(* CODESYS project Trabalho_final_v2.project

Project tree, tasks and I/O mapping:
  Device : CODESYS Control Win V3, 3S - Smart Software Solutions GmbH, order no. 305021, version 3.5.11.40
    application Application
      libraries: Standard, * (System)
      task MainTask (cyclic, interval t#20ms, priority 1) calls mode_selector, flow_controller, Automatic_Tank_Controller, CoolantLevelController, flow_controller, GinFlowController, RefrigeranteFlowController, TankLevelController_T1, TankLevelController_T2, TemperatureController, VermouthFlowController, SendProductController, ConveyorControl, TonelCounter, ProductInletControl, ProductSendControl, TonelLevelControl, MixerRotationControl
      global variables GVL
      program mode_selector [LD]
      program flow_controller [SFC]: MANUAL_active, AUTOMATICO_active
      program Automatic_Tank_Controller [SFC]: Colocar_gin_active, Colocar_verm_active, Ligar_motor_active, Resfriar_active, Tirar_refrige_active, Envio_T2_active, DESATIVAR_active, REINICIAR_T1_active, Limpar_T1_active
      program TankLevelController_T1 [ST]
      program TankLevelController_T2 [ST]
      program GinFlowController [ST]
      program VermouthFlowController [ST]
      program RefrigeranteFlowController [ST]
      program TemperatureController [ST]
      program CoolantLevelController [ST]
      program SendProductController [ST]
      program ConveyorControl [SFC]: Limpa_esteira_active, Liga_esteira_active, IN_PRODU_active, Inicio_active
      program TonelCounter [ST]
      program ProductInletControl [SFC]: RETIRA_ESTEIRA_active, ABRI_TORNE_active
      program ProductSendControl [ST]
      program TonelLevelControl [ST]
      program MixerRotationControl [ST]
*)

// Device/Application/GVL
{attribute 'qualified_only'}
VAR_GLOBAL
	

	// Ativação do sistema e escolha do modo
	Ligar : BOOL := FALSE;
	EMG : BOOL := FALSE;
	Sistema_ativo: BOOL;
	Seletor: BOOL;
	Selecionado: BOOL;
	Modo_manual: BOOL;
	Modo_automatico: BOOL;
	
	
	// Ativadores de modos
	Ativador_manual: BOOL := FALSE;
	Ativador_automatico: BOOL := FALSE;
	
	// Quantidades T1
	Quantidade_total_t1 : REAL := 0;
	
	// Indicadores T1
	Tanque01_vazio : BOOL;
	Tanque01_30L : BOOL;
	Tanque01_45L : BOOL;
	Tanque01_50L : BOOL;
	
	// Quantidades de bebida
	Quantidade_total_gin : REAL := 0;
	Quantidade_total_vermouth : REAL := 0;
	Quantidade_total_refrigerante : REAL := 0;
	
	// Temporizadores bebidas
	Temporizador_entrada_gin : TON;
	Temporizador_entrada_vermouth : TON;
	Temporizador_entrada_refrigerante : TON;
	Temporizador_saida_refrigerante : TON;
	Temporizador_resfriamento : TON;
	
	// Indicadores refrigerante
	Auto_nivel_refrigerante : BOOL := FALSE;
	Baixo_nivel_refrigerante : BOOL := TRUE;
	
	// Ativador temperatura
	Ativador_temperatura : BOOL := FALSE;
	
	// Indicadores de temperatura
	Temperatura_0c : BOOL := FALSE;
	Temperatura : REAL := 27;
	
	// Quantidade t2
	Quantidade_total_t2 : REAL := 0;
	
	// Indicadores T2
	Tanque02_vazio : BOOL;
	Tanque02_10p : BOOL;
	Tanque02_50p : BOOL;
	Tanque02_85p : BOOL;
	Tanque02_95p : BOOL;
	
	//valvulas T1
	Valvula_gin : BOOL := FALSE;
	Valvula_vermouth : BOOL := FALSE;
	Valvula_refrigerante : BOOL := FALSE;
	Valvula_descarte_refrigerante : BOOL := FALSE;
	
	//Temporizadores T1
	Temporizador_descarte_produto : TON;
	Temporizador_envio_produto : TON;
	
	// Instrumentos t1
	Motor_t1 : BOOL := FALSE;
	
	// Instrumentos entre t1 e t2
	Bomba : BOOL := FALSE;
	
	// valvulas entre tanques
	Valvula_entre_tanques : BOOL := FALSE;
	Valvula_descarte : BOOL := FALSE;
	Valvula_entrada_t2 : BOOL := FALSE;
	
	//Instrumentos t2
	Esteira : BOOL;
	Termino_envio: BOOL;
	
	
	// Contadores Toneis
	Numero_toneis_liberados : REAL;
	Numero_toneis_prduzidos : REAL;
	Numero_toneis_total : REAL;
	Tonel_produzido : BOOL;
	Total_tonel_menor4: BOOL;
	Total_tonel_4: BOOL;
	
	// Temporizador produção esteira
	Temporizador_producao_esteira : TON;
	
	// Controle para o envio de produto para os toneis
	Tonel_preparado : BOOL := FALSE;
	Tonel_cheio : BOOL;
	
	// VALVULAS T2 TONEL
	Valvula_t2_tonel : BOOL := FALSE;
	Temporizador_t2_tonel : TON;
	
	//Quantidade tonel
	Quantidade_tonel : REAL;
	
	Termino_tonel : BOOL;
	Sem_produto : BOOL;
	
	// Controladores do misturador
	TON_Partida : TON;
    TON_Parada : TON;
    M101_Partida_Em_Andamento : BOOL := FALSE;
    M101_Parada_Em_Andamento : BOOL := FALSE;
	DutyCycle_OUT : REAL := 0;
END_VAR

// Device/Application/mode_selector
PROGRAM mode_selector
VAR
END_VAR

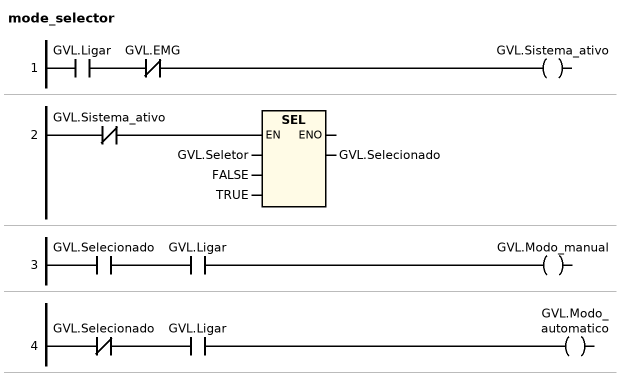
// NETWORK 1
GVL.Sistema_ativo := GVL.Ligar AND NOT GVL.EMG;

// NETWORK 2
IF NOT GVL.Sistema_ativo THEN GVL.Selecionado := SEL(GVL.Seletor, FALSE, TRUE); END_IF

// NETWORK 3
GVL.Modo_manual := GVL.Selecionado AND GVL.Ligar;

// NETWORK 4
GVL.Modo_automatico := NOT GVL.Selecionado AND GVL.Ligar;

END_PROGRAM

// Device/Application/flow_controller
PROGRAM flow_controller
VAR
END_VAR

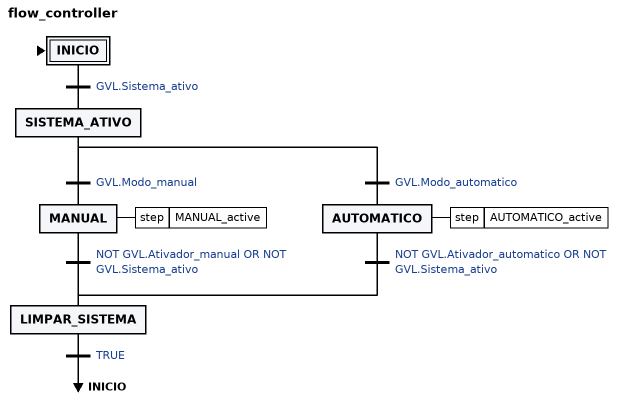
INITIAL_STEP INICIO:
END_STEP
TRANSITION FROM INICIO TO SISTEMA_ATIVO
    := GVL.Sistema_ativo;
END_TRANSITION
STEP SISTEMA_ATIVO:
END_STEP
TRANSITION FROM SISTEMA_ATIVO TO MANUAL
    := GVL.Modo_manual;
END_TRANSITION
STEP MANUAL:
    MANUAL_active(N);  // step action
END_STEP
TRANSITION FROM MANUAL TO LIMPAR_SISTEMA
    := NOT GVL.Ativador_manual OR NOT GVL.Sistema_ativo;
END_TRANSITION
TRANSITION FROM SISTEMA_ATIVO TO AUTOMATICO
    := GVL.Modo_automatico;
END_TRANSITION
STEP AUTOMATICO:
    AUTOMATICO_active(N);  // step action
END_STEP
TRANSITION FROM AUTOMATICO TO LIMPAR_SISTEMA
    := NOT GVL.Ativador_automatico OR NOT GVL.Sistema_ativo;
END_TRANSITION
STEP LIMPAR_SISTEMA:
END_STEP
TRANSITION FROM LIMPAR_SISTEMA TO INICIO
    := TRUE;
END_TRANSITION

ACTION MANUAL_active:
GVL.Ativador_manual := TRUE;
END_ACTION

ACTION AUTOMATICO_active:
GVL.Ativador_automatico := TRUE;
END_ACTION

END_PROGRAM

// Device/Application/Automatic_Tank_Controller
PROGRAM Automatic_Tank_Controller
VAR
END_VAR

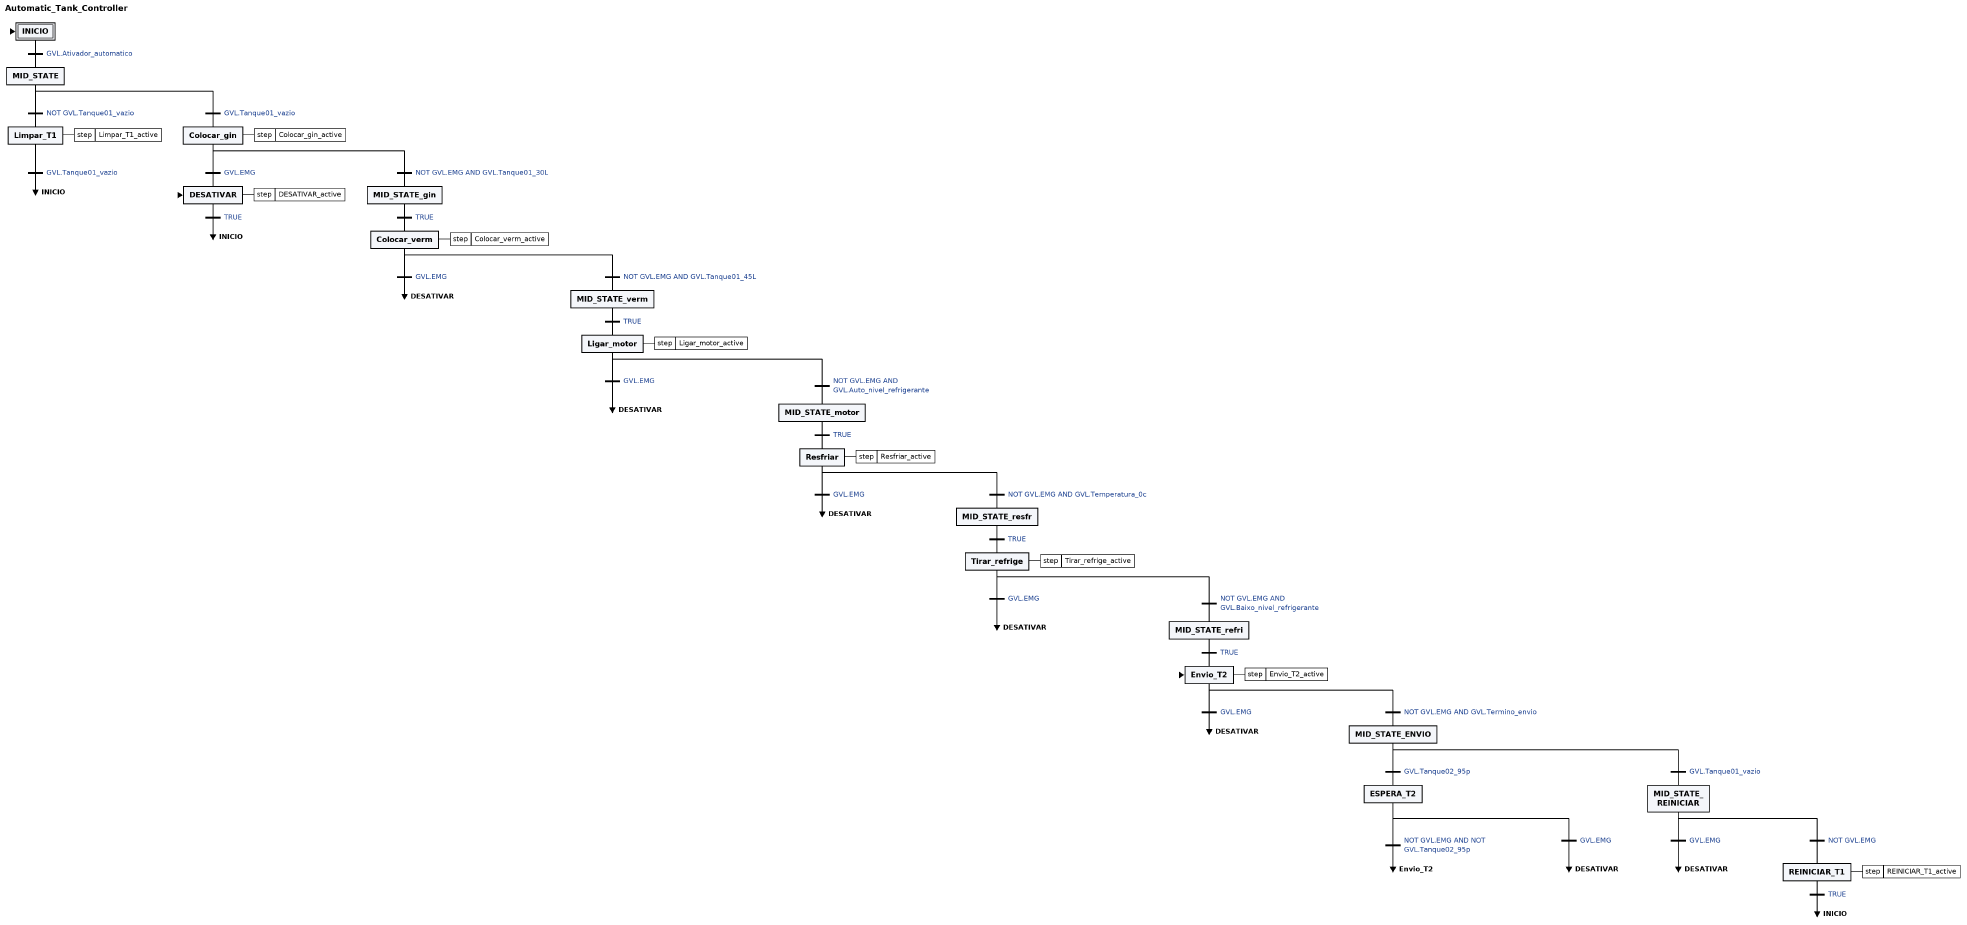
INITIAL_STEP INICIO:
END_STEP
TRANSITION FROM INICIO TO MID_STATE
    := GVL.Ativador_automatico;
END_TRANSITION
STEP MID_STATE:
END_STEP
TRANSITION FROM MID_STATE TO Limpar_T1
    := NOT GVL.Tanque01_vazio;
END_TRANSITION
STEP Limpar_T1:
    Limpar_T1_active(N);  // step action
END_STEP
TRANSITION FROM Limpar_T1 TO INICIO
    := GVL.Tanque01_vazio;
END_TRANSITION
TRANSITION FROM MID_STATE TO Colocar_gin
    := GVL.Tanque01_vazio;
END_TRANSITION
STEP Colocar_gin:
    Colocar_gin_active(N);  // step action
END_STEP
TRANSITION FROM Colocar_gin TO DESATIVAR
    := GVL.EMG;
END_TRANSITION
STEP DESATIVAR:
    DESATIVAR_active(N);  // step action
END_STEP
TRANSITION FROM DESATIVAR TO INICIO
    := TRUE;
END_TRANSITION
TRANSITION FROM Colocar_gin TO MID_STATE_gin
    := NOT GVL.EMG AND GVL.Tanque01_30L;
END_TRANSITION
STEP MID_STATE_gin:
END_STEP
TRANSITION FROM MID_STATE_gin TO Colocar_verm
    := TRUE;
END_TRANSITION
STEP Colocar_verm:
    Colocar_verm_active(N);  // step action
END_STEP
TRANSITION FROM Colocar_verm TO DESATIVAR
    := GVL.EMG;
END_TRANSITION
TRANSITION FROM Colocar_verm TO MID_STATE_verm
    := NOT GVL.EMG AND GVL.Tanque01_45L;
END_TRANSITION
STEP MID_STATE_verm:
END_STEP
TRANSITION FROM MID_STATE_verm TO Ligar_motor
    := TRUE;
END_TRANSITION
STEP Ligar_motor:
    Ligar_motor_active(N);  // step action
END_STEP
TRANSITION FROM Ligar_motor TO DESATIVAR
    := GVL.EMG;
END_TRANSITION
TRANSITION FROM Ligar_motor TO MID_STATE_motor
    := NOT GVL.EMG AND GVL.Auto_nivel_refrigerante;
END_TRANSITION
STEP MID_STATE_motor:
END_STEP
TRANSITION FROM MID_STATE_motor TO Resfriar
    := TRUE;
END_TRANSITION
STEP Resfriar:
    Resfriar_active(N);  // step action
END_STEP
TRANSITION FROM Resfriar TO DESATIVAR
    := GVL.EMG;
END_TRANSITION
TRANSITION FROM Resfriar TO MID_STATE_resfr
    := NOT GVL.EMG AND GVL.Temperatura_0c;
END_TRANSITION
STEP MID_STATE_resfr:
END_STEP
TRANSITION FROM MID_STATE_resfr TO Tirar_refrige
    := TRUE;
END_TRANSITION
STEP Tirar_refrige:
    Tirar_refrige_active(N);  // step action
END_STEP
TRANSITION FROM Tirar_refrige TO DESATIVAR
    := GVL.EMG;
END_TRANSITION
TRANSITION FROM Tirar_refrige TO MID_STATE_refri
    := NOT GVL.EMG AND GVL.Baixo_nivel_refrigerante;
END_TRANSITION
STEP MID_STATE_refri:
END_STEP
TRANSITION FROM MID_STATE_refri TO Envio_T2
    := TRUE;
END_TRANSITION
STEP Envio_T2:
    Envio_T2_active(N);  // step action
END_STEP
TRANSITION FROM Envio_T2 TO DESATIVAR
    := GVL.EMG;
END_TRANSITION
TRANSITION FROM Envio_T2 TO MID_STATE_ENVIO
    := NOT GVL.EMG AND GVL.Termino_envio;
END_TRANSITION
STEP MID_STATE_ENVIO:
END_STEP
TRANSITION FROM MID_STATE_ENVIO TO ESPERA_T2
    := GVL.Tanque02_95p;
END_TRANSITION
STEP ESPERA_T2:
END_STEP
TRANSITION FROM ESPERA_T2 TO Envio_T2
    := NOT GVL.EMG AND NOT GVL.Tanque02_95p;
END_TRANSITION
TRANSITION FROM ESPERA_T2 TO DESATIVAR
    := GVL.EMG;
END_TRANSITION
TRANSITION FROM MID_STATE_ENVIO TO MID_STATE_REINICIAR
    := GVL.Tanque01_vazio;
END_TRANSITION
STEP MID_STATE_REINICIAR:
END_STEP
TRANSITION FROM MID_STATE_REINICIAR TO DESATIVAR
    := GVL.EMG;
END_TRANSITION
TRANSITION FROM MID_STATE_REINICIAR TO REINICIAR_T1
    := NOT GVL.EMG;
END_TRANSITION
STEP REINICIAR_T1:
    REINICIAR_T1_active(N);  // step action
END_STEP
TRANSITION FROM REINICIAR_T1 TO INICIO
    := TRUE;
END_TRANSITION

ACTION Colocar_gin_active:
GVL.Valvula_gin := TRUE;
END_ACTION

ACTION Colocar_verm_active:
GVL.Valvula_vermouth := TRUE;
END_ACTION

ACTION Ligar_motor_active:
GVL.Motor_t1 := TRUE;
GVL.Valvula_refrigerante := TRUE;
END_ACTION

ACTION Resfriar_active:
GVL.Ativador_temperatura := TRUE;
END_ACTION

ACTION Tirar_refrige_active:
GVL.Motor_t1 := FALSE;
GVL.Valvula_descarte_refrigerante := TRUE;
END_ACTION

ACTION Envio_T2_active:
GVL.Valvula_entre_tanques := TRUE;
GVL.Bomba := TRUE;
GVL.Valvula_entrada_t2 := TRUE;
END_ACTION

ACTION DESATIVAR_active:
GVL.Ativador_automatico := FALSE;
END_ACTION

ACTION REINICIAR_T1_active:
GVL.Valvula_gin := FALSE;
GVL.Valvula_vermouth := FALSE;
GVL.Valvula_descarte_refrigerante := FALSE;
GVL.Valvula_refrigerante := FALSE;
GVL.Motor_t1 := FALSE;
GVL.Bomba := FALSE;
GVL.Temperatura := 27;
GVL.Quantidade_total_gin := 0;
GVL.Quantidade_total_vermouth := 0;
GVL.Quantidade_total_refrigerante := 0;
GVL.Temperatura_0c := FALSE;
END_ACTION

ACTION Limpar_T1_active:
GVL.Bomba := TRUE;
GVL.Valvula_entre_tanques := TRUE;
GVL.Valvula_descarte := TRUE;

IF GVL.Quantidade_total_t1 < 0 THEN
		GVL.Quantidade_total_t1 := 0;
		GVL.Bomba := FALSE;
		GVL.Valvula_entre_tanques := FALSE;
		GVL.Valvula_descarte := FALSE;
ELSE
	IF GVL.Quantidade_total_t1 > 0 THEN
		GVL.Temporizador_descarte_produto(IN:=TRUE, PT:=T#0.5S);
		IF GVL.Temporizador_descarte_produto.Q THEN
			GVL.Quantidade_total_t1 := GVL.Quantidade_total_t1 - 5;
		END_IF
	ELSE
		IF GVL.Quantidade_total_t1 = 0 THEN
			GVL.Bomba := FALSE;
			GVL.Valvula_entre_tanques := FALSE;
			GVL.Valvula_descarte := FALSE;
		END_IF
	END_IF
END_IF
END_ACTION

END_PROGRAM

// Device/Application/CoolantLevelController
PROGRAM CoolantLevelController
VAR
END_VAR

IF GVL.Quantidade_total_refrigerante = 0 THEN
	GVL.Baixo_nivel_refrigerante := TRUE;
	GVL.Auto_nivel_refrigerante := FALSE;
END_IF

IF GVL.Quantidade_total_refrigerante = 15 THEN
	GVL.Baixo_nivel_refrigerante := FALSE;
	GVL.Auto_nivel_refrigerante := TRUE;
END_IF

END_PROGRAM

// Device/Application/GinFlowController
PROGRAM GinFlowController
VAR
	Limite : REAL;
END_VAR

IF GVL.Modo_automatico THEN
	Limite := 30;
ELSE
	Limite := 52;
END_IF


IF NOT GVL.EMG AND GVL.Valvula_gin THEN
	IF GVL.Quantidade_total_gin < Limite THEN
		GVL.Temporizador_entrada_gin(IN:=TRUE, PT:=T#0.5S);
		IF GVL.Temporizador_entrada_gin.Q THEN
			GVL.Quantidade_total_gin := GVL.Quantidade_total_gin + 2;
			GVL.Quantidade_total_t1 := GVL.Quantidade_total_t1 + 2;
			GVL.Temporizador_entrada_gin(IN:=FALSE);
		END_IF
	ELSE
		GVL.Valvula_gin := FALSE;
	END_IF
END_IF

END_PROGRAM

// Device/Application/RefrigeranteFlowController
PROGRAM RefrigeranteFlowController
VAR
	Limite: REAL := 15;
END_VAR

IF NOT GVL.EMG AND GVL.Valvula_refrigerante THEN
	IF GVL.Quantidade_total_refrigerante <= Limite THEN 
		GVL.Temporizador_entrada_refrigerante(IN:=TRUE, PT:=T#0.5S);
		IF GVL.Temporizador_entrada_refrigerante.Q THEN
			GVL.Quantidade_total_refrigerante := GVL.Quantidade_total_refrigerante + 1.666;
			GVL.Temporizador_entrada_refrigerante(IN:=FALSE);
		END_IF
	ELSE
		GVL.Valvula_refrigerante := FALSE;
		GVL.Quantidade_total_refrigerante := 15;
	END_IF
END_IF


IF NOT GVL.EMG AND GVL.Valvula_descarte_refrigerante THEN
	IF GVL.Quantidade_total_refrigerante > 0 THEN 
		GVL.Temporizador_saida_refrigerante(IN:=TRUE, PT:=T#0.5S);
		IF GVL.Temporizador_saida_refrigerante.Q THEN
			GVL.Quantidade_total_refrigerante := GVL.Quantidade_total_refrigerante - 1.666;
			GVL.Temporizador_saida_refrigerante(IN:=FALSE);
		END_IF
	ELSE
		GVL.Valvula_descarte_refrigerante := FALSE;
		GVL.Quantidade_total_refrigerante := 0;
	END_IF
END_IF

END_PROGRAM

// Device/Application/TankLevelController_T1
PROGRAM TankLevelController_T1
VAR
END_VAR

IF GVL.Quantidade_total_t1 = 0 THEN
	GVL.Tanque01_vazio := TRUE;
	GVL.Tanque01_30L := FALSE;
	GVL.Tanque01_45L := FALSE;
	GVL.Tanque01_50L := FALSE;
	
ELSIF GVL.Quantidade_total_t1 = 30 THEN
	GVL.Tanque01_vazio := FALSE;
	GVL.Tanque01_30L := TRUE;
	GVL.Tanque01_45L := FALSE;
	GVL.Tanque01_50L := FALSE;
	
ELSIF GVL.Quantidade_total_t1 = 45 THEN
	GVL.Tanque01_vazio := FALSE;
	GVL.Tanque01_30L := FALSE;
	GVL.Tanque01_45L := TRUE;
	GVL.Tanque01_50L := FALSE;
	
ELSIF GVL.Quantidade_total_t1 = 50 THEN
	GVL.Tanque01_vazio := FALSE;
	GVL.Tanque01_30L := FALSE;
	GVL.Tanque01_45L := FALSE;
	GVL.Tanque01_50L := TRUE;
END_IF;

END_PROGRAM

// Device/Application/TankLevelController_T2
PROGRAM TankLevelController_T2
VAR
END_VAR

IF GVL.Quantidade_total_t2 = 0 THEN
    GVL.Tanque02_vazio := TRUE;
    GVL.Tanque02_10p := FALSE;
    GVL.Tanque02_50p := FALSE;
    GVL.Tanque02_85p := FALSE;
    GVL.Tanque02_95p := FALSE;
    
ELSIF GVL.Quantidade_total_t2 > 0 AND GVL.Quantidade_total_t2 < 20 THEN
    GVL.Tanque02_vazio := FALSE;
    GVL.Tanque02_10p := FALSE;
    GVL.Tanque02_50p := FALSE;
    GVL.Tanque02_85p := FALSE;
    GVL.Tanque02_95p := FALSE;
    
ELSIF GVL.Quantidade_total_t2 >= 20 AND GVL.Quantidade_total_t2 < 100 THEN
    GVL.Tanque02_vazio := FALSE;
    GVL.Tanque02_10p := TRUE;
    GVL.Tanque02_50p := FALSE;
    GVL.Tanque02_85p := FALSE;
    GVL.Tanque02_95p := FALSE;
    
ELSIF GVL.Quantidade_total_t2 >= 100 AND GVL.Quantidade_total_t2 < 170 THEN
    GVL.Tanque02_vazio := FALSE;
    GVL.Tanque02_10p := FALSE;
    GVL.Tanque02_50p := TRUE; 
    GVL.Tanque02_85p := FALSE;
    GVL.Tanque02_95p := FALSE;
    
ELSIF GVL.Quantidade_total_t2 >= 170 AND GVL.Quantidade_total_t2 < 190 THEN
    GVL.Tanque02_vazio := FALSE;
    GVL.Tanque02_10p := FALSE;
    GVL.Tanque02_50p := FALSE;
    GVL.Tanque02_85p := TRUE;
    GVL.Tanque02_95p := FALSE;
    
ELSIF GVL.Quantidade_total_t2 >= 190 THEN
    GVL.Tanque02_vazio := FALSE;
    GVL.Tanque02_10p := FALSE;
    GVL.Tanque02_50p := FALSE;
    GVL.Tanque02_85p := FALSE;
    GVL.Tanque02_95p := TRUE; 
END_IF

END_PROGRAM

// Device/Application/TemperatureController
PROGRAM TemperatureController
VAR
END_VAR

IF GVL.Quantidade_total_refrigerante = 15 AND GVL.Ativador_temperatura THEN
	IF GVL.Temperatura > 0 THEN
		GVL.Temporizador_resfriamento(IN := TRUE, PT:=T#1S);
		IF GVL.Temporizador_resfriamento.Q THEN
			GVL.Temperatura := GVL.Temperatura - 2;
			GVL.Temporizador_resfriamento(IN := FALSE);
		END_IF
	ELSE
		IF GVL.Temperatura = 0 THEN
			GVL.Temperatura_0c := TRUE;
			GVL.Ativador_temperatura := FALSE;
		ELSE
			IF GVL.Temperatura < 0 THEN
				GVL.Temperatura := 0;
			END_IF
		END_IF
	END_IF
END_IF

END_PROGRAM

// Device/Application/VermouthFlowController
PROGRAM VermouthFlowController
VAR
	Limite: REAL;
END_VAR

IF GVL.Modo_automatico THEN
	Limite := 15;
ELSE
	Limite := 52;
END_IF


IF NOT GVL.EMG AND GVL.Valvula_vermouth THEN
	IF GVL.Quantidade_total_vermouth < Limite THEN
		GVL.Temporizador_entrada_vermouth(IN:=TRUE, PT:=T#0.5S);
		IF GVL.Temporizador_entrada_vermouth.Q THEN
			GVL.Quantidade_total_vermouth := GVL.Quantidade_total_vermouth +  1.666;
			GVL.Quantidade_total_t1 := GVL.Quantidade_total_t1 +  1.666;
			GVL.Temporizador_entrada_vermouth(IN:=FALSE);
		END_IF
	ELSE
		GVL.Quantidade_total_vermouth := Limite;
		GVL.Quantidade_total_t1 := 45;
		GVL.Valvula_vermouth := FALSE;
	END_IF
END_IF

END_PROGRAM

// Device/Application/SendProductController
PROGRAM SendProductController
VAR
END_VAR

IF NOT GVL.EMG AND GVL.Bomba AND GVL.Valvula_entrada_t2 AND GVL.Valvula_entre_tanques THEN
	GVL.Termino_envio := FALSE;
	IF GVL.Tanque02_95p THEN
		GVL.Bomba := FALSE;
		GVL.Valvula_entre_tanques:=FALSE;
		GVL.Valvula_entrada_t2:=FALSE;
		GVL.Termino_envio := TRUE;
	ELSE
		IF GVL.Quantidade_total_t1 > 0 THEN
			GVL.Temporizador_envio_produto(IN:=TRUE, PT:=T#0.5S);
			IF GVL.Temporizador_envio_produto.Q THEN
				GVL.Quantidade_total_t1:= GVL.Quantidade_total_t1 - 5;
				GVL.Quantidade_total_t2:= GVL.Quantidade_total_t2 + 5;
				GVL.Temporizador_envio_produto(IN:=FALSE);
			END_IF
		ELSE
			GVL.Bomba := FALSE;
			GVL.Valvula_entre_tanques:=FALSE;
			GVL.Valvula_entrada_t2:=FALSE;
			GVL.Termino_envio := TRUE;
		END_IF
 	END_IF
END_IF

END_PROGRAM

// Device/Application/ConveyorControl
PROGRAM ConveyorControl
VAR
END_VAR

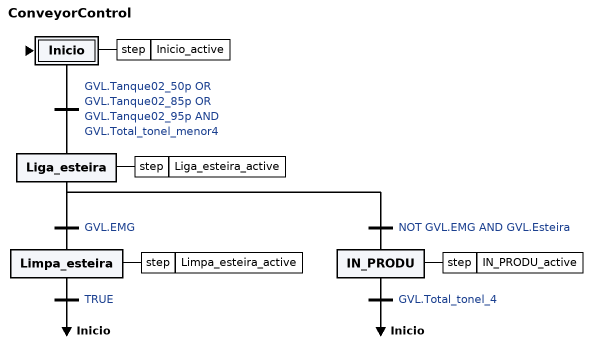
INITIAL_STEP Inicio:
    Inicio_active(N);  // step action
END_STEP
TRANSITION FROM Inicio TO Liga_esteira
    := GVL.Tanque02_50p OR GVL.Tanque02_85p OR GVL.Tanque02_95p AND GVL.Total_tonel_menor4;
END_TRANSITION
STEP Liga_esteira:
    Liga_esteira_active(N);  // step action
END_STEP
TRANSITION FROM Liga_esteira TO Limpa_esteira
    := GVL.EMG;
END_TRANSITION
STEP Limpa_esteira:
    Limpa_esteira_active(N);  // step action
END_STEP
TRANSITION FROM Limpa_esteira TO Inicio
    := TRUE;
END_TRANSITION
TRANSITION FROM Liga_esteira TO IN_PRODU
    := NOT GVL.EMG AND GVL.Esteira;
END_TRANSITION
STEP IN_PRODU:
    IN_PRODU_active(N);  // step action
END_STEP
TRANSITION FROM IN_PRODU TO Inicio
    := GVL.Total_tonel_4;
END_TRANSITION

ACTION Limpa_esteira_active:
GVL.Numero_toneis_liberados := 0;
GVL.Numero_toneis_prduzidos := 0;
GVL.Numero_toneis_total := 0;
GVL.Tonel_produzido := FALSE;
END_ACTION

ACTION Liga_esteira_active:
GVL.Esteira := TRUE;
GVL.Tonel_produzido := FALSE;
END_ACTION

ACTION IN_PRODU_active:
IF GVL.Numero_toneis_prduzidos < 4 AND GVL.Esteira THEN 
    GVL.Temporizador_producao_esteira(IN:=TRUE, PT:=T#15S);
    IF GVL.Temporizador_producao_esteira.Q THEN
        GVL.Numero_toneis_prduzidos := GVL.Numero_toneis_prduzidos + 1;
        GVL.Temporizador_producao_esteira(IN:=FALSE);
    END_IF
END_IF
END_ACTION

ACTION Inicio_active:
GVL.Tonel_produzido := TRUE;
GVL.Esteira := FALSE;
END_ACTION

END_PROGRAM

// Device/Application/TonelCounter
PROGRAM TonelCounter
VAR
END_VAR

IF GVL.Numero_toneis_prduzidos = 4 THEN
	GVL.Total_tonel_4 := TRUE;
	GVL.Total_tonel_menor4 := FALSE;
	GVL.Tonel_preparado := TRUE;
ELSE 
	IF GVL.Numero_toneis_prduzidos < 4 THEN
		GVL.Total_tonel_4 := FALSE;
		GVL.Total_tonel_menor4 := TRUE;
		GVL.Tonel_preparado := FALSE;
	END_IF
END_IF

END_PROGRAM

// Device/Application/ProductInletControl
PROGRAM ProductInletControl
VAR
END_VAR

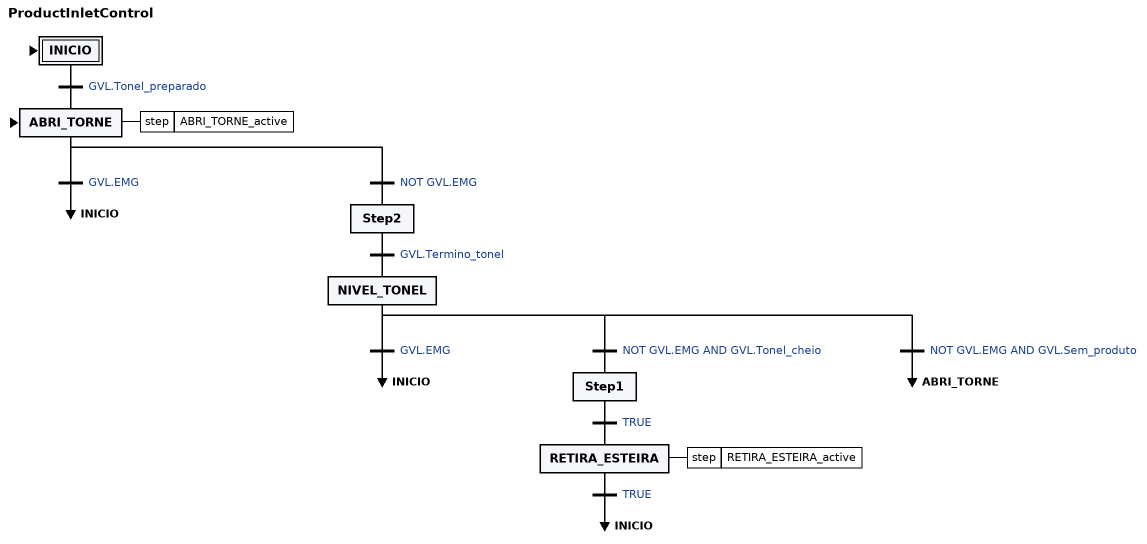
INITIAL_STEP INICIO:
END_STEP
TRANSITION FROM INICIO TO ABRI_TORNE
    := GVL.Tonel_preparado;
END_TRANSITION
STEP ABRI_TORNE:
    ABRI_TORNE_active(N);  // step action
END_STEP
TRANSITION FROM ABRI_TORNE TO INICIO
    := GVL.EMG;
END_TRANSITION
TRANSITION FROM ABRI_TORNE TO Step2
    := NOT GVL.EMG;
END_TRANSITION
STEP Step2:
END_STEP
TRANSITION FROM Step2 TO NIVEL_TONEL
    := GVL.Termino_tonel;
END_TRANSITION
STEP NIVEL_TONEL:
END_STEP
TRANSITION FROM NIVEL_TONEL TO INICIO
    := GVL.EMG;
END_TRANSITION
TRANSITION FROM NIVEL_TONEL TO Step1
    := NOT GVL.EMG AND GVL.Tonel_cheio;
END_TRANSITION
TRANSITION FROM NIVEL_TONEL TO ABRI_TORNE
    := NOT GVL.EMG AND GVL.Sem_produto;
END_TRANSITION
STEP Step1:
END_STEP
TRANSITION FROM Step1 TO RETIRA_ESTEIRA
    := TRUE;
END_TRANSITION
STEP RETIRA_ESTEIRA:
    RETIRA_ESTEIRA_active(N);  // step action
END_STEP
TRANSITION FROM RETIRA_ESTEIRA TO INICIO
    := TRUE;
END_TRANSITION

ACTION RETIRA_ESTEIRA_active:
GVL.Numero_toneis_liberados := GVL.Numero_toneis_liberados + 1;
GVL.Numero_toneis_prduzidos := GVL.Numero_toneis_prduzidos - 1;
GVL.Quantidade_tonel := 0;
GVL.Termino_tonel := FALSE;
GVL.Sem_produto := FALSE;
END_ACTION

ACTION ABRI_TORNE_active:
GVL.Valvula_t2_tonel := TRUE;
GVL.Termino_tonel:=FALSE;
END_ACTION

END_PROGRAM

// Device/Application/ProductSendControl
PROGRAM ProductSendControl
VAR
END_VAR

IF NOT GVL.EMG AND GVL.Valvula_t2_tonel THEN
	IF GVL.Quantidade_total_t2 >= 1 THEN
		IF GVL.Quantidade_tonel < 15 THEN
			GVL.Temporizador_t2_tonel(IN:=TRUE, PT:=T#0.5S);
			IF GVL.Temporizador_t2_tonel.Q THEN
				GVL.Quantidade_total_t2 := GVL.Quantidade_total_t2 - 1;
				GVL.Quantidade_tonel := GVL.Quantidade_tonel + 1;
				GVL.Temporizador_t2_tonel(IN:=FALSE);
			END_IF
		ELSE
			GVL.Valvula_t2_tonel := FALSE;
		END_IF
	ELSE
		GVL.Valvula_t2_tonel := FALSE;
		GVL.Sem_produto := TRUE;
	END_IF
	GVL.Termino_tonel:=TRUE;
END_IF

END_PROGRAM

// Device/Application/TonelLevelControl
PROGRAM TonelLevelControl
VAR
END_VAR

IF GVL.Quantidade_tonel = 15 THEN
	GVL.Tonel_cheio := TRUE;
ELSE
	GVL.Tonel_cheio := FALSE;
END_IF

END_PROGRAM

// Device/Application/MixerRotationControl
PROGRAM MixerRotationControl
VAR
END_VAR


// ----------------------------------------------------
// Lógica de Partida (0 a 100% em 5s)
// ----------------------------------------------------

// Inicia a partida quando o comando LIGAR é dado e não está desligando
IF GVL.Motor_t1 AND NOT GVL.M101_Partida_Em_Andamento AND NOT GVL.M101_Parada_Em_Andamento THEN
    GVL.M101_Partida_Em_Andamento := TRUE;
    GVL.TON_Partida(IN := TRUE, PT := T#5S); // Reinicia a contagem
ELSIF GVL.Motor_t1 AND GVL.M101_Partida_Em_Andamento THEN
    GVL.TON_Partida(IN := TRUE, PT := T#5S); // Mantém a contagem
ELSE
    GVL.TON_Partida(IN := FALSE, PT := T#5S); // Para a contagem se não estiver mais ligando
END_IF

// Cálculo do Duty Cycle durante a Partida
IF GVL.M101_Partida_Em_Andamento THEN
    GVL.DutyCycle_OUT := (TIME_TO_REAL(GVL.TON_Partida.ET) / TIME_TO_REAL(T#5S)) * 100.0;
    
    IF GVL.TON_Partida.Q THEN
        GVL.DutyCycle_OUT := 100.0; // Garante 100% no final da rampa
        GVL.M101_Partida_Em_Andamento := FALSE;
    END_IF
END_IF

// ----------------------------------------------------
// Lógica de Parada (100 a 0% em 10s)
// ----------------------------------------------------

// Inicia a parada quando o comando LIGAR é desativado
IF NOT GVL.Motor_t1 AND NOT GVL.M101_Parada_Em_Andamento AND GVL.DutyCycle_OUT > 0.0 THEN
    GVL.M101_Parada_Em_Andamento := TRUE;
    GVL.TON_Parada(IN := TRUE, PT := T#10S); // Reinicia a contagem de parada
ELSIF NOT GVL.Motor_t1 AND GVL.M101_Parada_Em_Andamento THEN
    GVL.TON_Parada(IN := TRUE, PT := T#10S); // Mantém a contagem
ELSE
    GVL.TON_Parada(IN := FALSE, PT := T#10S); // Para a contagem
END_IF

// Cálculo do Duty Cycle durante a Parada
IF GVL.M101_Parada_Em_Andamento THEN
    GVL.DutyCycle_OUT := 100.0 - ((TIME_TO_REAL(GVL.TON_Parada.ET) / TIME_TO_REAL(T#10S)) * 100.0);

    IF GVL.TON_Parada.Q THEN
        GVL.DutyCycle_OUT := 0.0; // Garante 0% no final da rampa
        GVL.M101_Parada_Em_Andamento := FALSE;
    END_IF
END_IF

// ----------------------------------------------------
// Estado Estável e Limites
// ----------------------------------------------------
IF GVL.Motor_t1 AND NOT GVL.M101_Partida_Em_Andamento THEN
    GVL.DutyCycle_OUT := 100.0; // Mantém 100% durante a operação normal
END_IF

IF NOT GVL.Motor_t1 AND NOT GVL.M101_Parada_Em_Andamento THEN
    GVL.DutyCycle_OUT := 0.0; // Mantém 0% quando desligado
END_IF

// Limite para evitar erros de ponto flutuante
IF GVL.DutyCycle_OUT < 0.0 THEN
    GVL.DutyCycle_OUT := 0.0;
ELSIF GVL.DutyCycle_OUT > 100.0 THEN
    GVL.DutyCycle_OUT := 100.0;
END_IF

END_PROGRAM
